// TIA Portal V17 export
// export: Created 2023-06-23T18:33:38.30576Z, ExportSetting WithDefaults, DisplayName Totally Integrated Automation Portal, DisplayVersion V17, DisplayName TIA Portal Openness, DisplayVersion V17, DisplayName TIA Portal Version Control Interface, DisplayVersion V17, DisplayName STEP 7 Professional, DisplayVersion V17, DisplayName STEP 7 Safety, DisplayVersion V17, DisplayName WinCC Advanced / Unified PC, DisplayVersion V17
VAR_GLOBAL   // PLC tag table "08_CT-2"
   "iCT-2" AT %I1.5 : Bool;
   "oCT-2s" AT %Q20.4 : Bool;
   "oCT-2f" AT %Q20.5 : Bool;
END_VAR
